FUNCTION_BLOCK Aux_Val1_QW (* Output service interface function block for word output data *)
  (* Description: Copyright (c) 2015, 2016 fortiss GmbH, HR Agrartechnik GmbH This program and the accompanying materials are made available under the terms of the Eclipse Public License 2.0 which is available at https://www.eclipse.org/legal/epl-2.0/ SPDX-License-Identifier: EPL-2.0 Supported auxiliary types: 0, 1, 2, 3, 4, 6, 11, 12, 13 *)
  (* Version 1.0, 2015-09-22, Gerd Kainz, fortiss GmbH, initial API and implementation and/or initial documentation *)
  (* Version 1.1, 2016-07-18, Alois Zoitl, fortiss GmbH *)
  PACKAGE isobus::UT::io::Auxiliary::OUT;
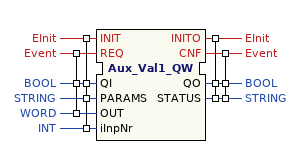
  EVENT_INPUT
    INIT : EInit WITH QI, PARAMS, iInpNr; (* Service Initialization *)
    REQ WITH QI, OUT; (* Service Request *)
  END_EVENT
  EVENT_OUTPUT
    INITO : EInit WITH QO, STATUS; (* Initialization Confirm *)
    CNF WITH QO, STATUS; (* Confirmation of Requested Service *)
  END_EVENT
  VAR_INPUT
    QI : BOOL; (* Event Input Qualifier *)
    PARAMS : STRING; (* Service Parameters *)
    OUT : WORD; (* Output data to resource *)
    iInpNr : INT := 0; (* Number of auxiliary array - corresponds with the order in the pool that means first aux input in pool is iInpNr = 0 etc. *)
  END_VAR
  VAR_OUTPUT
    QO : BOOL; (* Event Output Qualifier *)
    STATUS : STRING; (* Service Status *)
  END_VAR
END_FUNCTION_BLOCK
